FUNCTION_BLOCK FB_AssertResultStatic
VAR
    aAssertResults : ARRAY[1..cStartSizeOfArray] OF ST_AssertResult;
    nFailuresCount : UINT := 0;
    nSuccessCount : UINT := 0;
    nAssertTotalCount : UINT := 0;
END_VAR
VAR CONSTANT
    cStartSizeOfArray : UINT := 300;
END_VAR

(* This method searches for any already added additions of the combination of
   assertion message and assertion instance paths. It returns the location of
   the addition. If it is not found, it returns 0.
*)
METHOD PRIVATE FindMessageAndTestInstancePathEquals : UDINT
VAR_INPUT
    sMessage : Tc2_System.T_MaxString;
    sTestInstancePath : Tc2_System.T_MaxString;
END_VAR
VAR
    nCounter : UDINT;
END_VAR
FindMessageAndTestInstancePathEquals := 0;
IF nAssertTotalCount > 0 THEN
    FOR nCounter := 1 TO nAssertTotalCount BY 1 DO
        IF sMessage = aAssertResults[nCounter].sMessage AND
            sTestInstancePath = aAssertResults[nCounter].sTestInstancePath THEN
            FindMessageAndTestInstancePathEquals := nCounter;
            EXIT;
        END_IF
	END_FOR
END_IF
END_METHOD

METHOD PUBLIC ReportResult
VAR_INPUT
    Expected : ANY;
    Actual : ANY;
    sMessage : Tc2_System.T_MaxString;
    sTestInstancePath : Tc2_System.T_MaxString;
END_VAR
VAR_OUTPUT
    bAlreadyReported : BOOL := FALSE;
END_VAR
VAR
    nLocation : UDINT;
    bDataTypesNotEquals : BOOL;
    bDataSizeNotEquals : BOOL;
    bDataContentNotEquals : BOOL;
END_VAR
// Check if we can find any existing match of the report
IF (nLocation := FindMessageAndTestInstancePathEquals(sMessage, sTestInstancePath)) = 0 OR_ELSE
    (NOT F_IsAnyEqualToUnionValue(uExpectedOrActual := aAssertResults[nLocation].uExpected,
                                 ExpectedOrActual := Expected) OR
    NOT F_IsAnyEqualToUnionValue(uExpectedOrActual := aAssertResults[nLocation].uActual,
                                 ExpectedOrActual := Actual)) THEN

    // No existing match found, create a new entry
    F_AnyComparator(AnyValueOne := Expected,
                    AnyValueTwo := Actual,
                    bDataTypesNotEquals => bDataTypesNotEquals,
                    bDataSizeNotEquals => bDataSizeNotEquals,
                    bDataContentNotEquals => bDataContentNotEquals);

    IF bDataTypesNotEquals OR bDataSizeNotEquals OR bDataContentNotEquals THEN
        GVL_AssertResult.nAssertFailuresCount := GVL_AssertResult.nAssertFailuresCount + 1;
    ELSE
        GVL_AssertResult.nAssertSuccessCount := GVL_AssertResult.nAssertSuccessCount + 1;
	END_IF
    nAssertTotalCount := nAssertTotalCount + 1;
    aAssertResults[nAssertTotalCount].uExpected := F_AnyToUnionValue(AnyValue := Expected);
    aAssertResults[nAssertTotalCount].uActual := F_AnyToUnionValue(AnyValue := Actual);
    aAssertResults[nAssertTotalCount].sMessage := sMessage;
    aAssertResults[nAssertTotalCount].sTestInstancePath := sTestInstancePath;
ELSE
    bAlreadyReported := TRUE;
END_IF
END_METHOD

END_FUNCTION_BLOCK

(* stored: Version 1.1.0.1, ProductVersion 3.1.4022.12
   POU FB_AssertResultStatic: Id {9683a633-879e-475e-a97f-0742f9ecfd04}, SpecialFunc None
   Method FindMessageAndTestInstancePathEquals: Id {33a89dae-77cc-43e7-920d-ea254b349a40}
   Method ReportResult: Id {675e4dfe-54f1-4dc0-a6fd-481bc63973c5} *)
